// TIA Portal V17 export
// export: Created 2024-01-30T08:49:14.791955Z, ExportSetting WithDefaults, DisplayName Totally Integrated Automation Portal, DisplayVersion V17 Update 6, DisplayName TIA Portal Openness, DisplayVersion V17 Update 6, DisplayName TIA Portal Version Control Interface, DisplayVersion V17, DisplayName STEP 7 Professional, DisplayVersion V17 Update 6, DisplayName STEP 7 Safety, DisplayVersion V17 Update 6, DisplayName WinCC Advanced, DisplayVersion V17 Update 6
FUNCTION_BLOCK "B.01813_SIPP"   // FB7, LAD
{ S7_Optimized_Access := 'TRUE' }
VERSION : 0.1
// stored: AutoNumber true, IsIECCheckEnabled false, IsRetainMemResEnabled false, MemoryReserve 100, SetENOAutomatically false, UDAEnableTagReadback false
   VAR
      SQ_Activation_Time : UDInt;
      SQ_Act_time_inH : Real;
   END_VAR
BEGIN

REGION Network 1
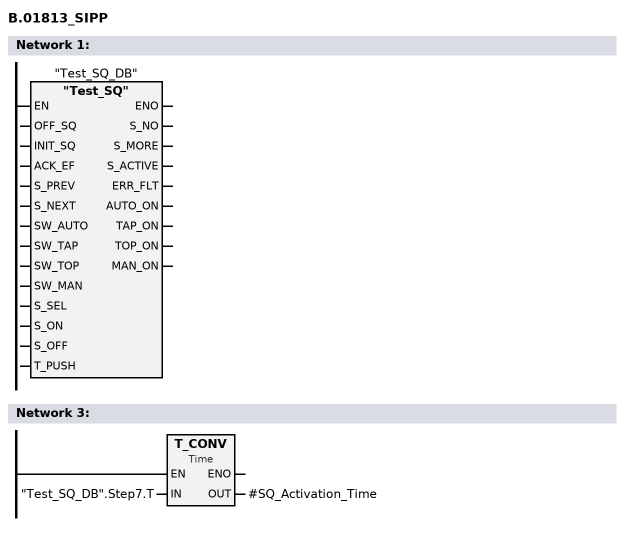
   RUNG wire#powerrail
      "Test_SQ_DB"(OFF_SQ :=, INIT_SQ :=, ACK_EF :=, S_PREV :=, S_NEXT :=, SW_AUTO :=, SW_TAP :=, SW_TOP :=, SW_MAN :=, S_SEL :=, S_ON :=, S_OFF :=, T_PUSH :=, S_NO =>, S_MORE =>, S_ACTIVE =>, ERR_FLT =>, AUTO_ON =>, TAP_ON =>, TOP_ON =>, MAN_ON =>)
   END_RUNG
   // the same network as SCL:
   "Test_SQ_DB"();   // "Test_SQ"
END_REGION

REGION Network 2 (SCL)
   #SQ_Act_time_inH := #SQ_Activation_Time / 1000.0 / 60 / 60;
END_REGION

REGION Network 3
   RUNG wire#powerrail
      { S7_Templates := "[src_type := Time, dest_type := UDInt]" } T_CONV(IN := "Test_SQ_DB".Step7.T, OUT => #SQ_Activation_Time)
   END_RUNG
   // the same network as SCL:
   T_CONV(IN := "Test_SQ_DB".Step7.T, OUT => #SQ_Activation_Time);
END_REGION
END_FUNCTION_BLOCK
